Universal Robots PolyScope program: AG_until_io.urp

Program AG_until_io (installation=AutoGrind directory=/programs/AutoGrind createdIn=5.9.1.1031110 lastSavedIn=5.9.1.1031110 robotSerialNumber=20195501059)
Calibrated DH parameters: a=[0.000146, -0.418764, -0.053981, 0.000058, -0.000023, 0]; d=[0.162545, 37.319448, -206.067439, 168.881546, 0.09955, 0.099464]; alpha=[1.57004, -0.001979, 0.002304, 1.570607, -1.57066, 0]; deltaTheta=[0, -0.174616, -1.258233, 1.432844, -0.000001, 0]
Robot Program (runOnlyOnce=true)
  MoveL speed 250 mm/s, acceleration 1200 mm/s^2 (useActiveTCP=true) feature=Base
    Waypoint Waypoint_1: TCP in base x=85.902 y=-446.434 z=70.228 mm, rx=-3.1319 ry=-0.0015 rz=0.0135 rad; joints [84.138, -86.15, 124.035, -127.377, -90.485, 174.117] deg; TCP offset x=0 y=0 z=175 mm, rx=0 ry=0 rz=0 rad
    MoveDirectionNode (selectedDirection=ZPlus toolParams=0.02, 0.4) feature=Joint_6_name
      Until IO (allowActions=false ioType=DIGITAL_INPUT digitalValue=false) pin=digital_in[3]
      Until TOOL_CONTACT_DETECTION (allowActions=false retraction=0.004 decelerationAcceleration=0.5 decelerationAngularAcceleration=34.906585)
    Waypoint Waypoint_1: TCP in base x=85.902 y=-446.434 z=70.228 mm, rx=-3.1319 ry=-0.0015 rz=0.0135 rad; joints [84.138, -86.15, 124.035, -127.377, -90.485, 174.117] deg
